PROGRAM MAIN
VAR
	test : ServoNC;
	
	home : BOOL;
	
	target : LREAL;
	
	pos, neg : BOOL;
END_VAR

test();

test.bEnable := TRUE;

IF NOT test.HomeSet THEN
	test.homingSequence();
	RETURN;
END_IF

test.stop();

IF pos THEN
	test.moveContinuous(direction := MC_Positive_Direction);
END_IF

IF neg THEN
	test.moveContinuous(direction := MC_Negative_Direction);
END_IF

IF target > -1000 AND target < -10 THEN
	test.moveAbsolute(newTarget := target);
END_IF

END_PROGRAM

(* stored: Version 1.1.0.1, ProductVersion 3.1.4024.11
   POU MAIN: Id {e81a1fb7-6f36-470e-826c-e121b98d210e}, SpecialFunc None *)
